{attribute 'qualified_only'}

TYPE machineDisplayStates :
(
	dStStartUp             := 10,
	dStEMGButtonDown,
	dStOpenDoors,
	dStNoAirSupplay,
	dStStationError,
	dStMachineIsStopping,
	dStMachineIsStopped,
	dStAutoRun,
	dStMachineStandBy,
	dStMachinePurgeActive
	
)DINT;
END_TYPE

(* stored: Version 1.1.0.1, ProductVersion 3.1.4024.3
   DUT machineDisplayStates: Id {aa42c474-de05-4380-aed2-5dd31752712f} *)
